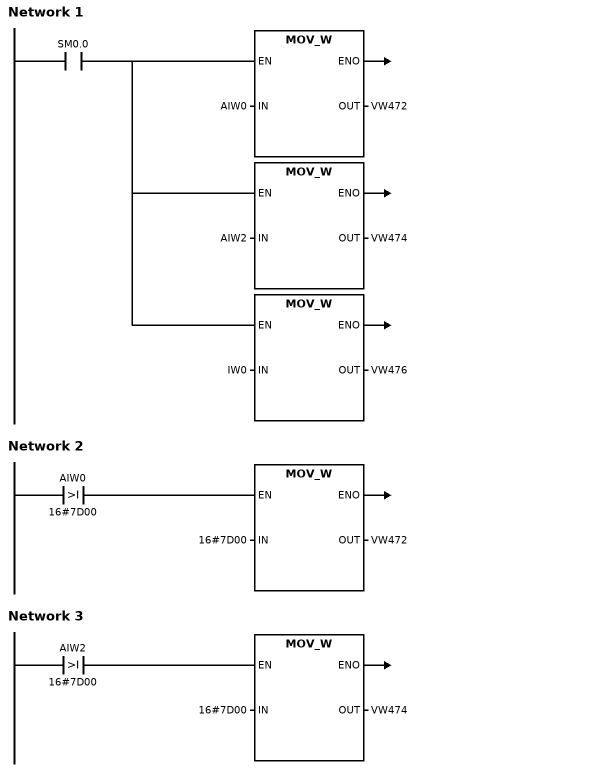
[picture p24: SBR19 networks 1-3]
Network 1
LD     SM0.0
MOVW   AIW0, VW472
MOVW   AIW2, VW474
MOVW   IW0, VW476
Network 2
LDW>   AIW0, 16#7D00
MOVW   16#7D00, VW472
Network 3
LDW>   AIW2, 16#7D00
MOVW   16#7D00, VW474
END_SUBROUTINE_BLOCK

INTERRUPT_BLOCK INT_0:INT0
TITLE=中断程序注释
BEGIN
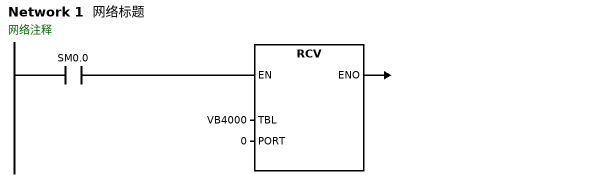
Network 1 // 网络标题
// 网络注释
LD     SM0.0
RCV    VB4000, 0
END_INTERRUPT_BLOCK

// INT1: protected block, not included

// INT2: protected block, not included

// INT3: protected block, not included

INTERRUPT_BLOCK INT_2:INT5
TITLE=
BEGIN
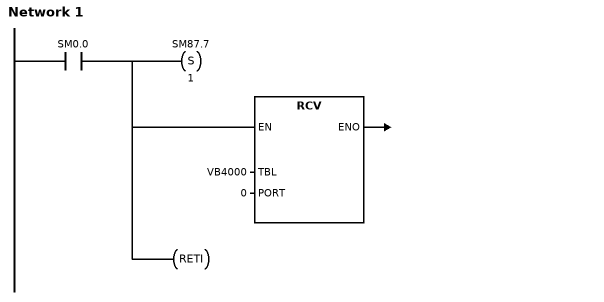
Network 1
LD     SM0.0
S      SM87.7, 1
RCV    VB4000, 0
CRETI
END_INTERRUPT_BLOCK
